(* IEC 61131-3 sources: Industry-PLC-LLM/data/PLCBEAD_repo/PLCBEAD_PLCEmbed-main/PLC-BEAD/Source/GEB/DATE_TO_UDINT, 1 file *)

(* ---- DATE_TO_UDINT.ST ---- *)
FUNCTION DATE_TO_UDINT2:UDINT
	VAR_INPUT
		IN :	UDINT;
	END_VAR

	DATE_TO_UDINT2 := IN;
END_FUNCTION

PROGRAM program0
  VAR
    LocalVar0 : UDINT;
	LocalOUT  : UDINT;
  END_VAR
  	LocalOUT := DATE_TO_UDINT2(LocalVar0);
END_PROGRAM
